(* Schneider Machine Expert - Basic project trying counter, file version 2.7.0.0 *)
(* ProjectInformations: Name=New project *)

HARDWARE
  Cpu 0: TM221M16R/G
  EthernetConfiguration: NetworkName=M221, IpAllocationMode=FixedAddress, IpAddress=0.0.0.0, SubnetMask=0.0.0.0
  SerialLineConfiguration: Baud=Baud19200, Parity=ParityEven, DataBits=DataBits8, StopBits=StopBits1, PhysicalMedium=PhysicalMediumRs485, TransmissionMode=TransmissionModeModbusRtu, SlaveId=1, Addressing=SlaveAddressing
  MastTask: UsePeriodScanMode=false, PeriodScan=100
  FastTask: Period=255
  CpuBehavior: StartingMode=StartAsPreviousState, AutoSaveRamOnEeprom=true, WatchdogPeriod=250

SYMBOLS  (address, symbol, comment, settings)
  %M0       RESET
  %M1       SET
  %M2       COUNT_UP
  %M3       COUNT_DOWN
  %M4       DOWN_COUNT_OVERFLOW
  %M5       PRESET_REACHED
  %M6       UP_COUNT_OVERFLOW
  %MW0      COUNTER_PRESET
  %MW1      COUNTER_VALUE

POU New POU
  (* SectionNumber=1 *)

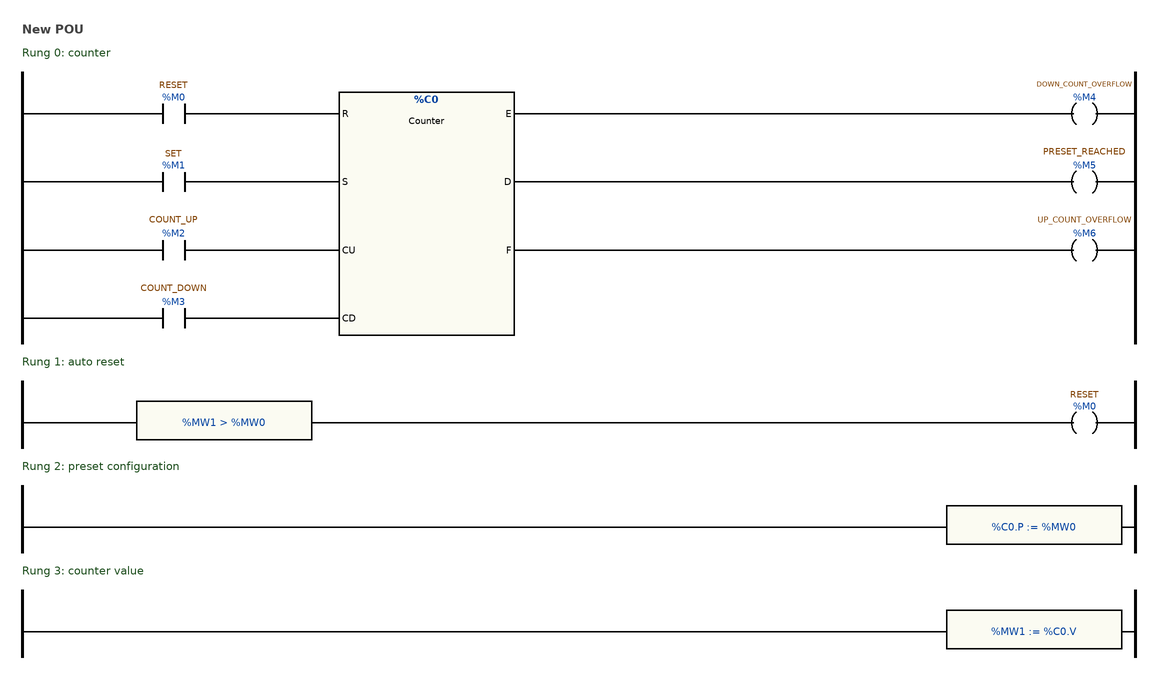

// Rung 0: counter
  BLK %C0
  LD %M0                  (* RESET *)
  R
  LD %M1                  (* SET *)
  S
  LD %M2                  (* COUNT_UP *)
  CU
  LD %M3                  (* COUNT_DOWN *)
  CD
  OUT_BLK
  LD E
  ST %M4                  (* DOWN_COUNT_OVERFLOW *)
  LD D
  ST %M5                  (* PRESET_REACHED *)
  LD F
  ST %M6                  (* UP_COUNT_OVERFLOW *)
  END_BLK
  // as ST:
  //   %C0(R := RESET, S := SET, CU := COUNT_UP, CD := COUNT_DOWN);
  //   DOWN_COUNT_OVERFLOW := %C0.E;
  //   PRESET_REACHED := %C0.D;
  //   UP_COUNT_OVERFLOW := %C0.F;

// Rung 1: auto reset
  LD 1
  AND [ %MW1 > %MW0 ]     (* COUNTER_VALUE, COUNTER_PRESET *)
  ST %M0                  (* RESET *)
  // as ST:
  //   RESET := COUNTER_VALUE > COUNTER_PRESET;

// Rung 2: preset configuration
  LD 1
  [ %C0.P := %MW0 ]       (* COUNTER_PRESET *)
  // as ST:
  //   %C0.P := COUNTER_PRESET;

// Rung 3: counter value
  LD 1
  [ %MW1 := %C0.V ]       (* COUNTER_VALUE *)
  // as ST:
  //   COUNTER_VALUE := %C0.V;
